FUNCTION_BLOCK FB_Test2
VAR_INPUT
END_VAR
VAR_OUTPUT
END_VAR
VAR
END_VAR

END_FUNCTION_BLOCK

(* stored: Version 1.1.0.1, ProductVersion 3.1.4024.10
   POU FB_Test2: Id {b41aa80a-a2e4-481a-87ef-3c1bfe538f57}, SpecialFunc None *)
